TYPE stKeyenceInspectionParams :
STRUCT
	bInspectionEnable	: BOOL;
	iMaxTrigRepeats		: INT 	:= 3;
	iProgramNumber		: UINT	:= 0;
END_STRUCT
END_TYPE

(* stored: Version 1.1.0.1, ProductVersion 3.1.4024.13
   DUT stKeyenceInspectionParams: Id {038c986d-b902-430c-a44c-895c36495da3} *)
